// TIA Portal V17 export
// export: Created 2025-03-07T09:17:08.550048Z, ExportSetting WithDefaults, DisplayName Totally Integrated Automation Portal, DisplayVersion V17 Update 8, DisplayName TIA Portal Openness, DisplayVersion V17 Update 8, DisplayName TIA Portal Version Control Interface, DisplayVersion V17, DisplayName SINAMICS Startdrive Advanced, DisplayVersion V17 SP2, DisplayName SINAMICS Startdrive G110M, G120, G120C, G120D, G120P, G115D, DisplayVersion V17 SP2, DisplayName SINAMICS Startdrive G130, G150, S120, S150, SINAMICS MV, S210, DisplayVersion V17 SP2, DisplayName STEP 7 Professional, DisplayVersion V17 Update 8, DisplayName SINUMERIK ONE STEP 7 Toolbox, DisplayVersion V17 Update 12, DisplayName SINUMERIK 840D sl STEP 7 Toolbox, DisplayVersion V17 Update 12, DisplayName STEP 7 Safety, DisplayVersion V17 Update 6, DisplayName WinCC Advanced, DisplayVersion V17 Update 8
FUNCTION_BLOCK "FB331_M_CODE_EXTENDED"   // FB331, LAD
{ S7_Optimized_Access := 'FALSE' }
AUTHOR : ETXETAR
VERSION : 1.0
// stored: AutoNumber false, IsIECCheckEnabled false, SetENOAutomatically false, UDAEnableTagReadback false
   VAR_INPUT
      NC_Chan_Num_Chan : Int;   // Channel Number to monitoring
   END_VAR
   VAR DB_SPECIFIC
      INDEX : Int;
      M_code : Array[100..999] of Bool;   // EXTENDED M CODE
   END_VAR
   VAR_TEMP
      TEMP0 : Int;
      DB_Channel : Int;
      Inst_DB : Int;
   END_VAR
BEGIN

NETWORK
TITLE = READ DATA / Data block for monitoring channel

//DB from channel
      L     #NC_Chan_Num_Chan;
      +     20;
      T     #DB_Channel;
//set DB instance assigned to FB
      L     DINO;
      T     #Inst_DB;
      NOP   0;

NETWORK
TITLE = Reset signal from M Code
      LAR1  P#0.0;
      L     900;
R001: T     #TEMP0;
      OPN   DB [#Inst_DB];
      A     "M_ONE";
      R     DBX [AR1, P#4.0];
      +AR1  P#0.1;
      L     #TEMP0;
      LOOP  R001;

NETWORK
TITLE = Set signal from "M function 1 (DInt)"
      OPN   DB [#DB_Channel];
      A     %DBX58.0;  // M function 1 change
      JCN   END1;

      LAR1  P#0.0;
      L     100;
      T     #INDEX;
      L     900;
S001: T     #TEMP0;

      L     %DBW72;
      L     #INDEX;
      ==I;
      JC    Mse1;
      L     #INDEX;
      +     1;
      T     #INDEX;
      +AR1  P#0.1;
      L     #TEMP0;
      LOOP  S001;
      JU    END1;
Mse1: OPN   DB [#Inst_DB];
      S     DBX [AR1, P#4.0];

END1: NOP   0;

NETWORK
TITLE = Set signal from "M function 2 (DInt)"
      OPN   DB [#DB_Channel];
      A     %DBX58.1;  // M function 2 change
      JCN   END2;

      LAR1  P#0.0;
      L     100;
      T     #INDEX;
      L     900;
S002: T     #TEMP0;

      L     %DBW78;
      L     #INDEX;
      ==I;
      JC    Mse2;
      L     #INDEX;
      +     1;
      T     #INDEX;
      +AR1  P#0.1;
      L     #TEMP0;
      LOOP  S002;
      JU    END2;
Mse2: OPN   DB [#Inst_DB];
      S     DBX [AR1, P#4.0];

END2: NOP   0;

NETWORK
TITLE = Set signal from "M function 3 (DInt)"
      OPN   DB [#DB_Channel];
      A     %DBX58.2;  // M function 3 change
      JCN   END3;

      LAR1  P#0.0;
      L     100;
      T     #INDEX;
      L     900;
S003: T     #TEMP0;

      L     %DBW84;
      L     #INDEX;
      ==I;
      JC    Mse3;
      L     #INDEX;
      +     1;
      T     #INDEX;
      +AR1  P#0.1;
      L     #TEMP0;
      LOOP  S003;
      JU    END3;
Mse3: OPN   DB [#Inst_DB];
      S     DBX [AR1, P#4.0];

END3: NOP   0;

NETWORK
TITLE = Set signal from "M function 4 (DInt)"
      OPN   DB [#DB_Channel];
      A     %DBX58.3;  // M function 4 change
      JCN   END4;

      LAR1  P#0.0;
      L     100;
      T     #INDEX;
      L     900;
S004: T     #TEMP0;

      L     %DBW90;
      L     #INDEX;
      ==I;
      JC    Mse4;
      L     #INDEX;
      +     1;
      T     #INDEX;
      +AR1  P#0.1;
      L     #TEMP0;
      LOOP  S004;
      JU    END4;
Mse4: OPN   DB [#Inst_DB];
      S     DBX [AR1, P#4.0];

END4: NOP   0;

NETWORK
TITLE = Set signal from "M function 5 (DInt)"
      OPN   DB [#DB_Channel];
      A     %DBX58.4;  // M function 5 change
      JCN   END5;

      LAR1  P#0.0;
      L     100;
      T     #INDEX;
      L     900;
S005: T     #TEMP0;

      L     %DBW96;
      L     #INDEX;
      ==I;
      JC    Mse5;
      L     #INDEX;
      +     1;
      T     #INDEX;
      +AR1  P#0.1;
      L     #TEMP0;
      LOOP  S005;
      JU    END5;
Mse5: OPN   DB [#Inst_DB];
      S     DBX [AR1, P#4.0];

END5: NOP   0;

NETWORK
TITLE = 
      BE;

END_FUNCTION_BLOCK
